INTERFACE IACEdge EXTENDS IACObject

PROPERTY AllocatedByFunction : IPAProcessFunction
GET
END_GET
SET
END_SET
END_PROPERTY

// Compares if ACUrl of Source and Target are identical
METHOD Compare : BOOL
VAR_INPUT
	edge : IACEdge;
END_VAR
END_METHOD

PROPERTY ConnectionType : ConnectionTypesEnum
GET
END_GET
END_PROPERTY

PROPERTY Source : IACPoint
GET
END_GET
END_PROPERTY

PROPERTY Target : IACPoint
GET
END_GET
END_PROPERTY

END_INTERFACE

(* stored: Version 1.1.0.1, ProductVersion 3.1.4020.12
   Itf IACEdge: Id {275672f9-5da1-4662-9ceb-1a8c0a230248}
   Property AllocatedByFunction: Id {b23122c8-d680-4243-9824-8c73c3ca439b}
   Get Get: Id {ffc248f3-0ab8-4ba1-b745-b135991e3db1}
   Set Set: Id {d516871a-8a02-4aaa-b31b-6ac8fe18a37a}
   Method Compare: Id {8f599827-1d85-4b21-97c1-d4d3d442b8de}
   Property ConnectionType: Id {97f6f5f6-5d9d-4ea2-af64-cf31eba61941}
   Get Get: Id {14101126-fc95-4728-aceb-95b4f283449e}
   Property Source: Id {76887e3e-2c6f-4e57-ac22-d10b745bfb29}
   Get Get: Id {f97f4c70-786d-4662-922f-b232a32bca28}
   Property Target: Id {734ec446-9d1d-444c-9e50-7bb21def4724}
   Get Get: Id {b35b772c-15ef-4a32-8481-f5c24c0c02ec} *)
